(* Logix 5000 project; controller DC01 vendor 1 type 14 code 165 rev 32.12; software revision 32.04; part 7 of 13 *)
(* tags used below, declared in another part *)
   CurrentSchedule : UDT_ShiftString_Breakdown;
   DC1_to_LN02_Messages : DINT[20];
   LN02_Main_Messages : DINT[250];
   LN02_MainLine_MSG_Out : MESSAGE;
   LN02_Schedule : UDT_Current_Status;
   LN02_Theoretical_Units_Counter : COUNTER;
   LN02EHM11 : DINT;
   LN02EJM02 : DINT;
   LN02EJM03 : DINT;
   LN02EKM01 : DINT;
   LN02EKM02 : DINT;
   LN02EKM03 : DINT;
   LN02ELM01 : DINT;
   LN02ELM02 : DINT;
   LN02ELM03 : DINT;
   LN02ELM04 : DINT;
   LN02ELM05 : DINT;
   LN02EMM01 : DINT;
   LN02EMM02 : DINT;
   LN02EMM03 : DINT;
   LN02SKS06 : DINT;
   LN02WHM09 : DINT;
   LN02WHM10 : DINT;
   LN02WJS01 : DINT;
   LN02WJS02 : DINT;
   LN02WJS03 : DINT;
   LN02WKM01 : DINT;
   LN02WKS01 : DINT;
   LN02WKS02 : DINT;
   LN02WKS03 : DINT;
   LN02WKS04 : DINT;
   LN02WKS05 : DINT;
   LN02WLM06 : DINT;
   LN02WLM07 : DINT;
   LN02WMM02 : DINT;
   LN02WMM03 : DINT;
   LN03_DataFromDC1 : DINT[20];
   LN03_Main_Messages : DINT[250];
   LN03_Schedule : UDT_Current_Status;
   LN03_ScheduleUnits_Produced_from_line : DINT;
   LN03_Weekly_Schedule : UDT_Weekly_Schedule;
(* LN02, continued *)

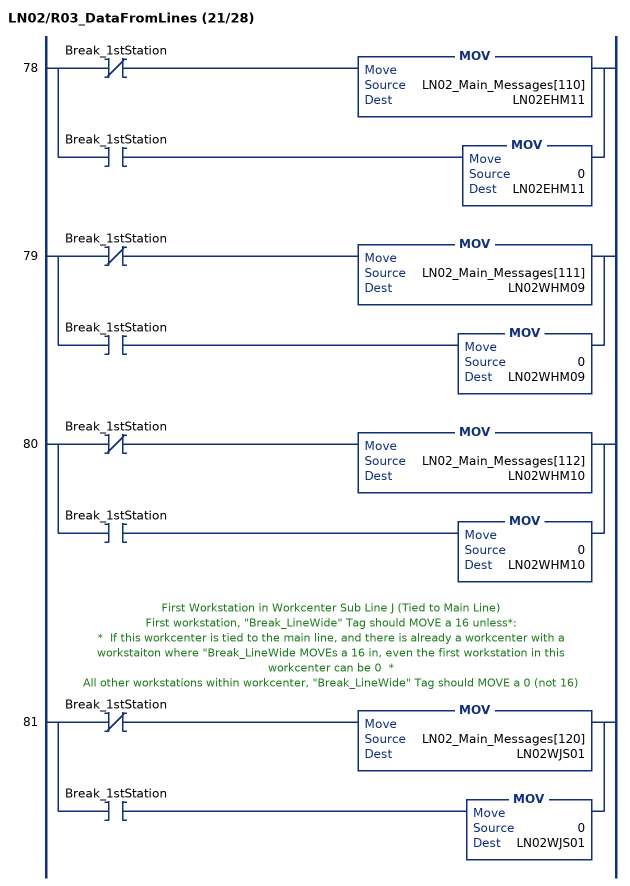
   78: [XIO(Break_1stStation) MOV(LN02_Main_Messages[110],LN02EHM11) ,XIC(Break_1stStation) MOV(0,LN02EHM11) ];
   79: [XIO(Break_1stStation) MOV(LN02_Main_Messages[111],LN02WHM09) ,XIC(Break_1stStation) MOV(0,LN02WHM09) ];
   80: [XIO(Break_1stStation) MOV(LN02_Main_Messages[112],LN02WHM10) ,XIC(Break_1stStation) MOV(0,LN02WHM10) ];
   // First Workstation in Workcenter Sub Line J (Tied to Main Line)
   // First workstation, "Break_LineWide" Tag should MOVE a 16 unless*:
   // *  If this workcenter is tied to the main line, and there is already a workcenter with a workstaiton where "Break_LineWide MOVEs a 16 in, even the first workstation in this workcenter can be 0  *
   // All other workstations within workcenter, "Break_LineWide" Tag should MOVE a 0 (not 16)
   81: [XIO(Break_1stStation) MOV(LN02_Main_Messages[120],LN02WJS01) ,XIC(Break_1stStation) MOV(0,LN02WJS01) ];
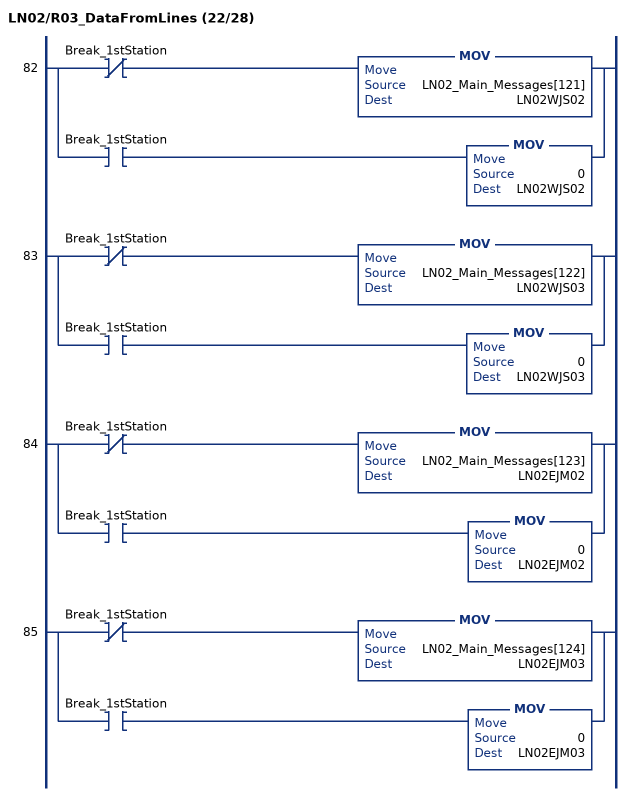
   82: [XIO(Break_1stStation) MOV(LN02_Main_Messages[121],LN02WJS02) ,XIC(Break_1stStation) MOV(0,LN02WJS02) ];
   83: [XIO(Break_1stStation) MOV(LN02_Main_Messages[122],LN02WJS03) ,XIC(Break_1stStation) MOV(0,LN02WJS03) ];
   84: [XIO(Break_1stStation) MOV(LN02_Main_Messages[123],LN02EJM02) ,XIC(Break_1stStation) MOV(0,LN02EJM02) ];
   85: [XIO(Break_1stStation) MOV(LN02_Main_Messages[124],LN02EJM03) ,XIC(Break_1stStation) MOV(0,LN02EJM03) ];
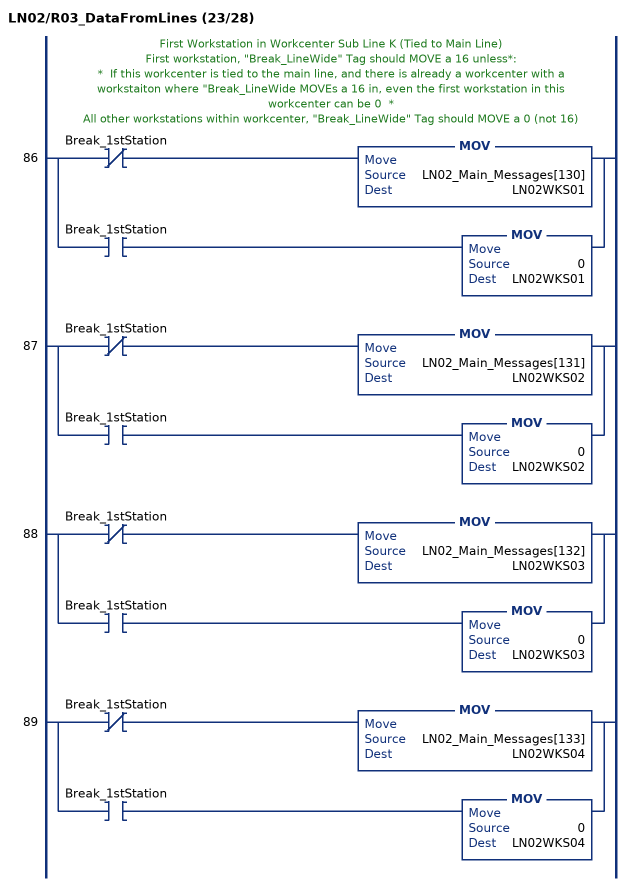
   // First Workstation in Workcenter Sub Line K (Tied to Main Line)
   // First workstation, "Break_LineWide" Tag should MOVE a 16 unless*:
   // *  If this workcenter is tied to the main line, and there is already a workcenter with a workstaiton where "Break_LineWide MOVEs a 16 in, even the first workstation in this workcenter can be 0  *
   // All other workstations within workcenter, "Break_LineWide" Tag should MOVE a 0 (not 16)
   86: [XIO(Break_1stStation) MOV(LN02_Main_Messages[130],LN02WKS01) ,XIC(Break_1stStation) MOV(0,LN02WKS01) ];
   87: [XIO(Break_1stStation) MOV(LN02_Main_Messages[131],LN02WKS02) ,XIC(Break_1stStation) MOV(0,LN02WKS02) ];
   88: [XIO(Break_1stStation) MOV(LN02_Main_Messages[132],LN02WKS03) ,XIC(Break_1stStation) MOV(0,LN02WKS03) ];
   89: [XIO(Break_1stStation) MOV(LN02_Main_Messages[133],LN02WKS04) ,XIC(Break_1stStation) MOV(0,LN02WKS04) ];
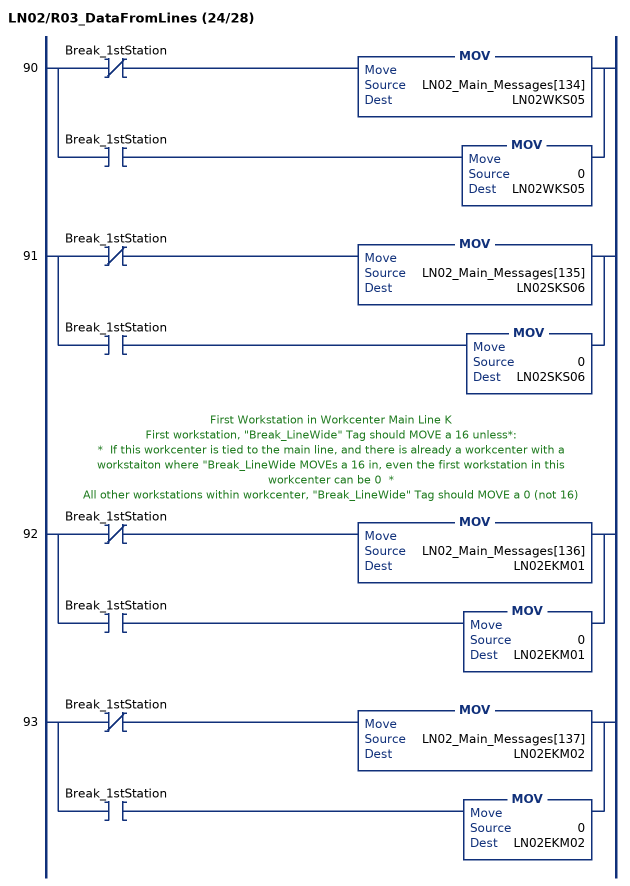
   90: [XIO(Break_1stStation) MOV(LN02_Main_Messages[134],LN02WKS05) ,XIC(Break_1stStation) MOV(0,LN02WKS05) ];
   91: [XIO(Break_1stStation) MOV(LN02_Main_Messages[135],LN02SKS06) ,XIC(Break_1stStation) MOV(0,LN02SKS06) ];
   // First Workstation in Workcenter Main Line K
   // First workstation, "Break_LineWide" Tag should MOVE a 16 unless*:
   // *  If this workcenter is tied to the main line, and there is already a workcenter with a workstaiton where "Break_LineWide MOVEs a 16 in, even the first workstation in this workcenter can be 0  *
   // All other workstations within workcenter, "Break_LineWide" Tag should MOVE a 0 (not 16)
   92: [XIO(Break_1stStation) MOV(LN02_Main_Messages[136],LN02EKM01) ,XIC(Break_1stStation) MOV(0,LN02EKM01) ];
   93: [XIO(Break_1stStation) MOV(LN02_Main_Messages[137],LN02EKM02) ,XIC(Break_1stStation) MOV(0,LN02EKM02) ];
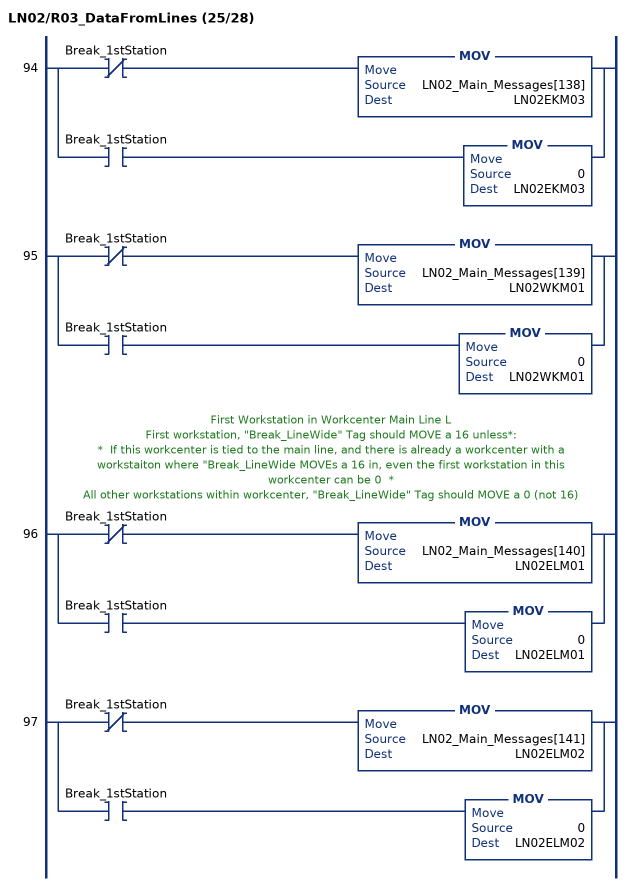
   94: [XIO(Break_1stStation) MOV(LN02_Main_Messages[138],LN02EKM03) ,XIC(Break_1stStation) MOV(0,LN02EKM03) ];
   95: [XIO(Break_1stStation) MOV(LN02_Main_Messages[139],LN02WKM01) ,XIC(Break_1stStation) MOV(0,LN02WKM01) ];
   // First Workstation in Workcenter Main Line L
   // First workstation, "Break_LineWide" Tag should MOVE a 16 unless*:
   // *  If this workcenter is tied to the main line, and there is already a workcenter with a workstaiton where "Break_LineWide MOVEs a 16 in, even the first workstation in this workcenter can be 0  *
   // All other workstations within workcenter, "Break_LineWide" Tag should MOVE a 0 (not 16)
   96: [XIO(Break_1stStation) MOV(LN02_Main_Messages[140],LN02ELM01) ,XIC(Break_1stStation) MOV(0,LN02ELM01) ];
   97: [XIO(Break_1stStation) MOV(LN02_Main_Messages[141],LN02ELM02) ,XIC(Break_1stStation) MOV(0,LN02ELM02) ];
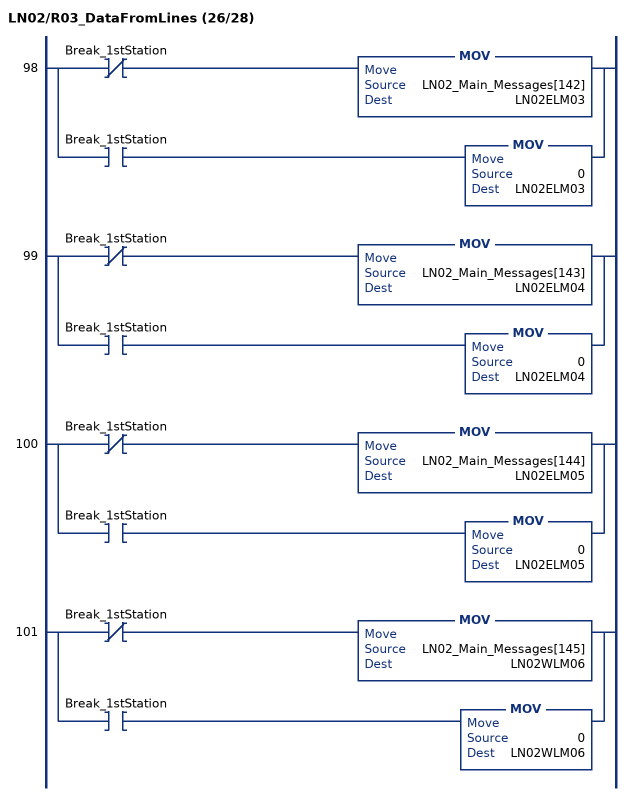
   98: [XIO(Break_1stStation) MOV(LN02_Main_Messages[142],LN02ELM03) ,XIC(Break_1stStation) MOV(0,LN02ELM03) ];
   99: [XIO(Break_1stStation) MOV(LN02_Main_Messages[143],LN02ELM04) ,XIC(Break_1stStation) MOV(0,LN02ELM04) ];
   100: [XIO(Break_1stStation) MOV(LN02_Main_Messages[144],LN02ELM05) ,XIC(Break_1stStation) MOV(0,LN02ELM05) ];
   101: [XIO(Break_1stStation) MOV(LN02_Main_Messages[145],LN02WLM06) ,XIC(Break_1stStation) MOV(0,LN02WLM06) ];
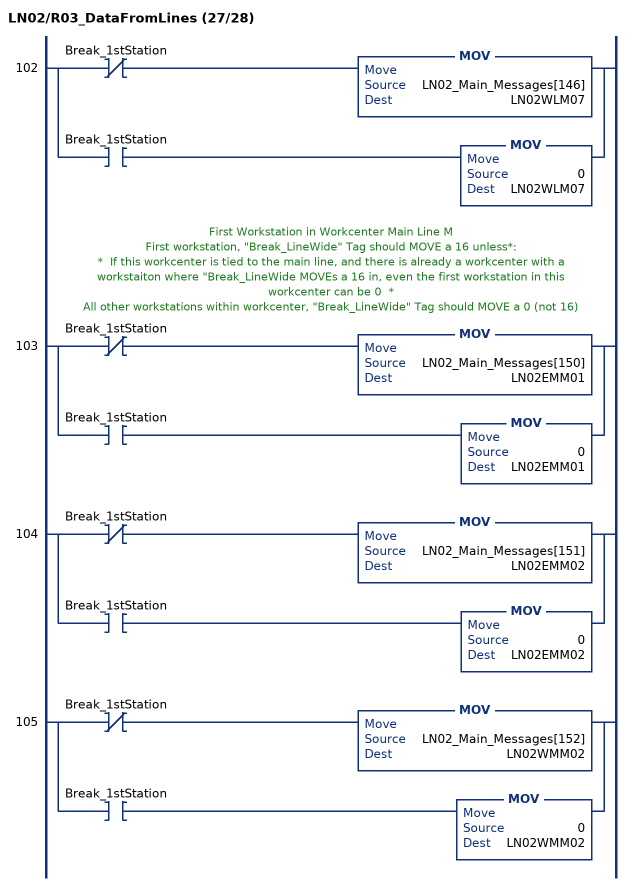
   102: [XIO(Break_1stStation) MOV(LN02_Main_Messages[146],LN02WLM07) ,XIC(Break_1stStation) MOV(0,LN02WLM07) ];
   // First Workstation in Workcenter Main Line M
   // First workstation, "Break_LineWide" Tag should MOVE a 16 unless*:
   // *  If this workcenter is tied to the main line, and there is already a workcenter with a workstaiton where "Break_LineWide MOVEs a 16 in, even the first workstation in this workcenter can be 0  *
   // All other workstations within workcenter, "Break_LineWide" Tag should MOVE a 0 (not 16)
   103: [XIO(Break_1stStation) MOV(LN02_Main_Messages[150],LN02EMM01) ,XIC(Break_1stStation) MOV(0,LN02EMM01) ];
   104: [XIO(Break_1stStation) MOV(LN02_Main_Messages[151],LN02EMM02) ,XIC(Break_1stStation) MOV(0,LN02EMM02) ];
   105: [XIO(Break_1stStation) MOV(LN02_Main_Messages[152],LN02WMM02) ,XIC(Break_1stStation) MOV(0,LN02WMM02) ];
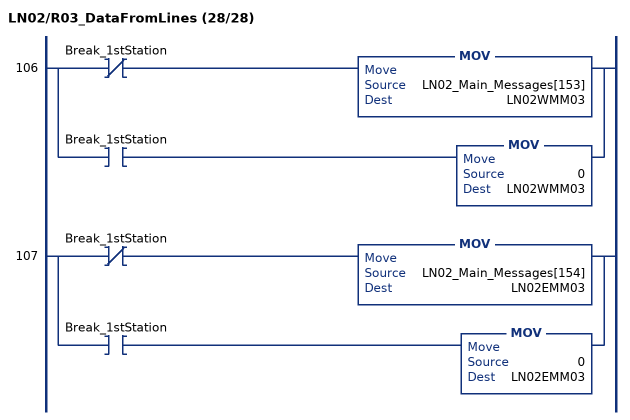
   106: [XIO(Break_1stStation) MOV(LN02_Main_Messages[153],LN02WMM03) ,XIC(Break_1stStation) MOV(0,LN02WMM03) ];
   107: [XIO(Break_1stStation) MOV(LN02_Main_Messages[154],LN02EMM03) ,XIC(Break_1stStation) MOV(0,LN02EMM03) ];
END_ROUTINE

ROUTINE R04_DataToLines   (* ladder *)
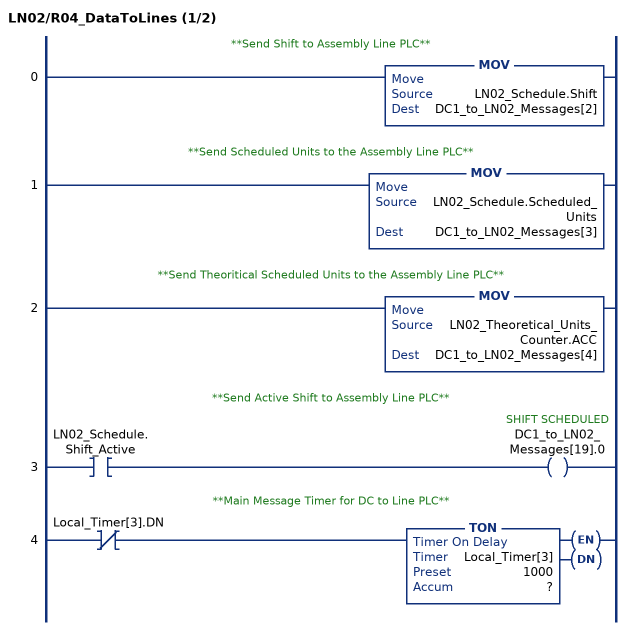
   // **Send Shift to Assembly Line PLC**
   0: MOV(LN02_Schedule.Shift,DC1_to_LN02_Messages[2]);
   // **Send Scheduled Units to the Assembly Line PLC**
   1: MOV(LN02_Schedule.Scheduled_Units,DC1_to_LN02_Messages[3]);
   // **Send Theoritical Scheduled Units to the Assembly Line PLC**
   2: MOV(LN02_Theoretical_Units_Counter.ACC,DC1_to_LN02_Messages[4]);
   // **Send Active Shift to Assembly Line PLC**
   3: XIC(LN02_Schedule.Shift_Active)OTE(DC1_to_LN02_Messages[19].0);
   // **Main Message Timer for DC to Line PLC**
   4: XIO(Local_Timer[3].DN)TON(Local_Timer[3],?,?);
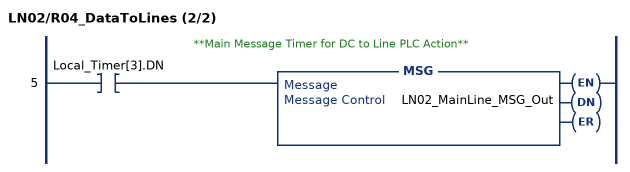
   // **Main Message Timer for DC to Line PLC Action**
   5: XIC(Local_Timer[3].DN)MSG(LN02_MainLine_MSG_Out);
END_ROUTINE
END_PROGRAM

PROGRAM LN03   (* main routine MainRoutine *)
VAR
   Always_Off : BOOL;
   Average_Array : DINT[20];
   Average_Sum : DINT;
   Averaged_LineSpeed : REAL;
   badModel : STRING_40;
   BlockStarveLocal : DINT;
   Break1_Hour : DINT;
   Break1_Hour_String : STRING;
   Break1_Length : DINT;
   Break1_MilliRemain : DINT;
   Break1_Min : DINT;
   Break1_Min_String : STRING;
   Break1_MinDisplay : DINT;
   Break1_SecDisplay : DINT;
   Break1_SecRemain : DINT;
   Break1_SecWholeMin : DINT;
   Break1_Timer : TIMER;
   Break2_Hour : DINT;
   Break2_Hour_String : STRING;
   Break2_Length : DINT;
   Break2_MilliRemain : DINT;
   Break2_Min : DINT;
   Break2_Min_String : STRING;
   Break2_MinDisplay : DINT;
   Break2_SecDisplay : DINT;
   Break2_SecRemain : DINT;
   Break2_SecWholeMin : DINT;
   Break2_Timer : TIMER;
   Break_1stStation : BOOL;
   Break_LineWide : BOOL;
   Break_WorkCenter : BOOL;
   Break_Workstation : BOOL;
   dlw_test : DINT := -805278210;
   End_Hour : DINT := 20;
   End_Hour_String : STRING := '20';
   End_Min : DINT := 3;
   End_Min_String : STRING := '3-';
   faultcount : DINT;
   FaultExists : CONTROL := (LEN := 230, POS := 229, EN := 1, DN := 1);
   firstCharacter : STRING_40 := 'W';
   FlexTimer_HoursDisplay : DINT;
   FlexTimer_MinutesDisplay : DINT;
   FlexTimer_SecondsDisplay : DINT;
   FlexTimertoHours : DINT;
   FlexTimertoMinutes : DINT;
   FlexTimertoSeconds : DINT;
   HoursFromMidnight : DINT;
   HoursFromMidnight_Remain : DINT;
   HoursTilMidnight : DINT;
   HoursTilMidnight_Remain : DINT;
   KnownFaultExist : DINT := 5;
   L02EAS35 : DINT;
   L02EDM16 : DINT;
   LineRate_perSecond_scheduled : DINT;
   LN01_Flex_Timer : TIMER;
   LN01_MainLine_MSG : MESSAGE;
        MessageParameters(ServiceCode := 16#004c, LocalElement := LN03_Main_Messages[0], ...)
   LN01_ML_Message_MSG : MESSAGE;
   LN01_Rotate_Timer : TIMER;
   LN01_SNModel_MSG : MESSAGE;
   LN02EAS35 : DINT;
   LN02EDM16 : DINT;
   LN03_MainLine_MSG : MESSAGE;   // Data Messages From Assembly Line 3 To Data Concentrator 1
        MessageParameters(ServiceCode := 16#004c, LocalElement := LN03_Main_Messages[0], ...)
   Local_Counter : COUNTER[20] := ([0].PRE := 1);
   Local_DATETIME : DINT[20];
   Local_Timer : TIMER[30] := ([0].EN := 1, [0].DN := 1, [3].PRE := 2000, [3].ACC := 1751, [3].EN := 1, [3].TT := 1, [4].PRE := 400, [4].ACC := 391, [4].EN := 1, [4].TT := 1, [6].PRE := 2000, [6].ACC := 150, [6].EN := 1, [6].TT := 1);
   Lunch_Hour : DINT;
   Lunch_Hour_String : STRING;
   Lunch_Length : DINT;
   Lunch_MilliRemain : DINT;
   Lunch_Min : DINT;
   Lunch_Min_String : STRING;
   Lunch_MinDisplay : DINT;
   Lunch_SecDisplay : DINT;
   Lunch_SecRemain : DINT;
   Lunch_SecWholeMin : DINT;
   Lunch_Timer : TIMER;
   Midnight_Hour : DINT;
   mlc_test21 : BOOL;
   null : STRING;
   OneShot : DINT;
   ONS_0 : DINT;
   ONS_20 : DINT;
   prevCalculateLocal : DINT;
   PreviousCount : DINT := 277;
   previousSerialNumber : STRING := 'CA0807422';
   PreviousShift : DINT := 1;
   readIndex : DINT := 41;
   register : DINT := 8;
   Rotate_MilliRemain : DINT;
   Rotate_Seconds_perShift : DINT;
   Rotate_SecRemain : DINT;
   Scheduled_Units_Buffer : DINT := 700;
   Shift_Break_Lengths : DINT;
   Shift_Break_Lengths_Remain : DINT;
   Shift_Delay_Min : DINT := 60;
   Shift_Extra_Min : DINT;
   Shift_Hours : DINT;
   Shift_Hours_Remain : DINT;
   Shift_Minutes : DINT;
   Shift_Minutes_Remain : DINT;
   Shift_Reset : BOOL;
   Shift_Reset_ONS : BOOL := 1;
   Shift_Seconds : DINT;
   Shift_Seconds_Remain : DINT;
   Start_Hour : DINT := 20;
   Start_Hour_String : STRING := '20';
   Start_Min : DINT := 3;
   Start_Min_String : STRING := '3-';
   tempIndex : DINT := 25;
   theoreticalUnitsReal : DINT;
   workstationid : DINT := 250;
   writeIndex : DINT := 42;
END_VAR

ROUTINE MainRoutine   (* ladder *)
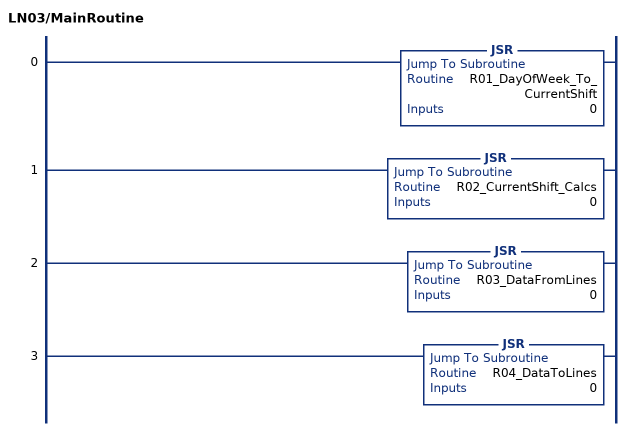
   0: JSR(R01_DayOfWeek_To_CurrentShift,0);
   1: JSR(R02_CurrentShift_Calcs,0);
   2: JSR(R03_DataFromLines,0);
   3: JSR(R04_DataToLines,0);
END_ROUTINE

ROUTINE R01_DayOfWeek_To_CurrentShift   (* ladder *)
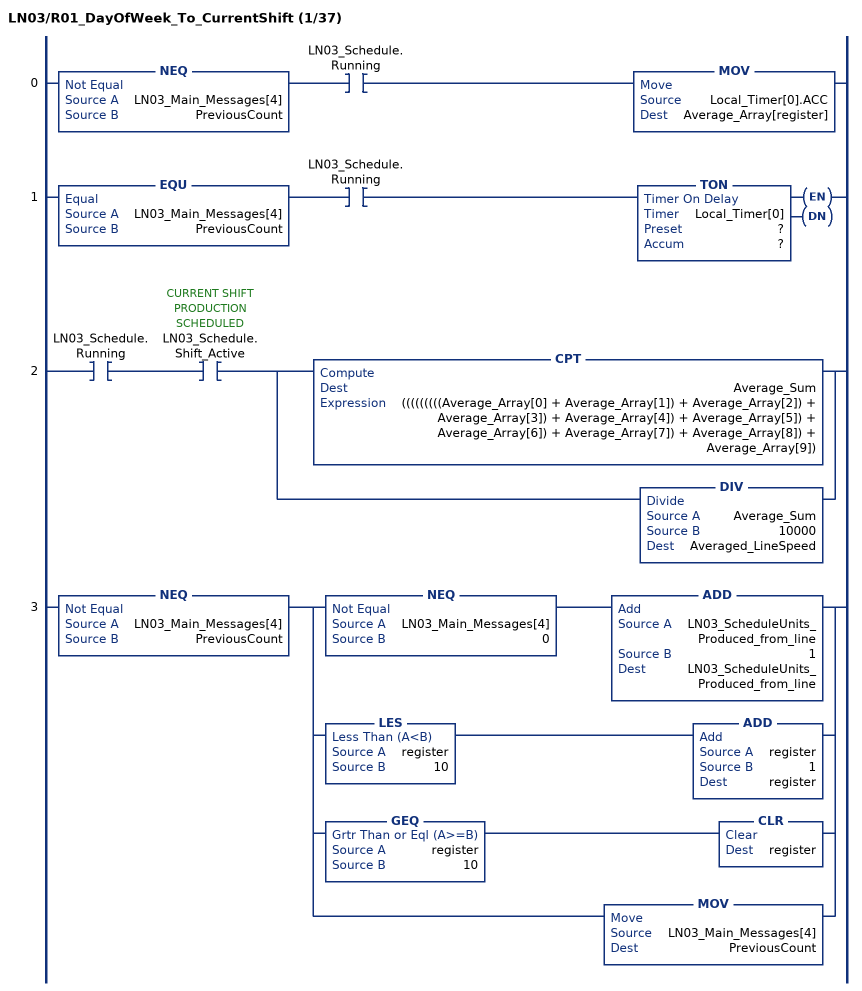
   0: NEQ(LN03_Main_Messages[4],PreviousCount)XIC(LN03_Schedule.Running)MOV(Local_Timer[0].ACC,Average_Array[register]);
   1: EQU(LN03_Main_Messages[4],PreviousCount)XIC(LN03_Schedule.Running)TON(Local_Timer[0],?,?);
   2: XIC(LN03_Schedule.Running)XIC(LN03_Schedule.Shift_Active)[CPT(Average_Sum,(((((((((Average_Array[0] + Average_Array[1]) + Average_Array[2]) + Average_Array[3]) + Average_Array[4]) + Average_Array[5]) + Average_Array[6]) + Average_Array[7]) + Average_Array[8]) + Average_Array[9])) ,DIV(Average_Sum,10000,Averaged_LineSpeed) ];
   3: NEQ(LN03_Main_Messages[4],PreviousCount)[NEQ(LN03_Main_Messages[4],0) ADD(LN03_ScheduleUnits_Produced_from_line,1,LN03_ScheduleUnits_Produced_from_line) ,LES(register,10) ADD(register,1,register) ,GEQ(register,10) CLR(register) ,MOV(LN03_Main_Messages[4],PreviousCount) ];
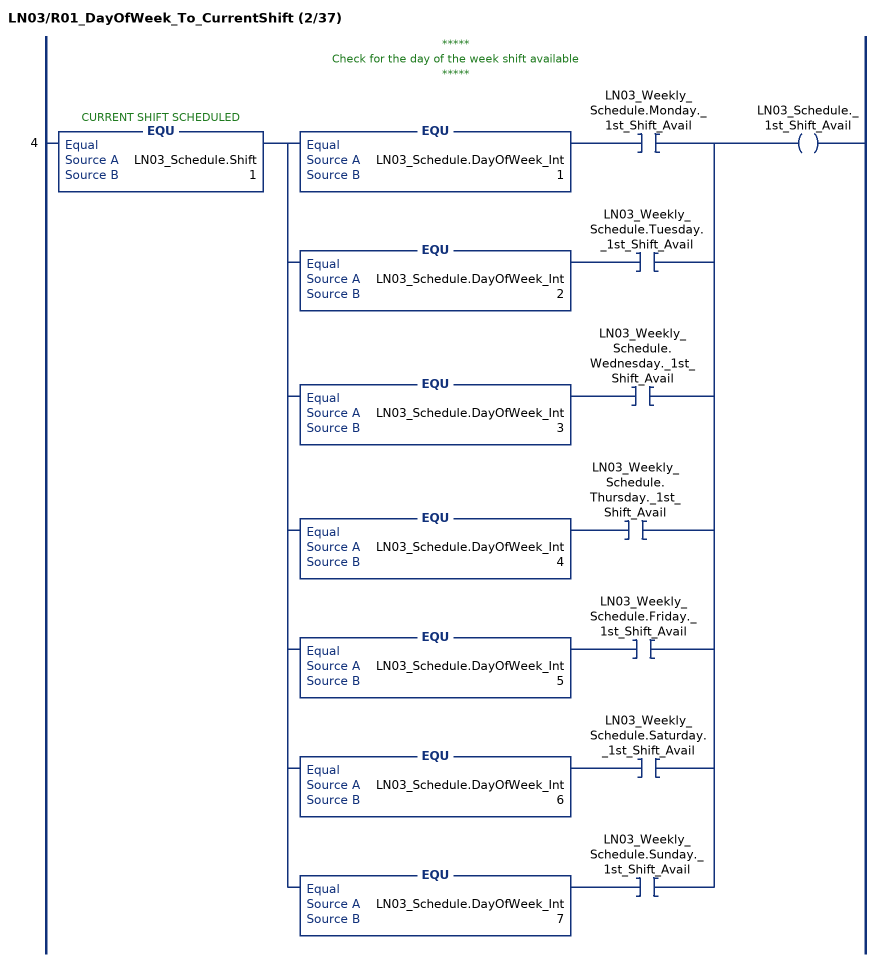
   // *****
   // Check for the day of the week shift available
   // *****
   4: EQU(LN03_Schedule.Shift,1)[EQU(LN03_Schedule.DayOfWeek_Int,1) XIC(LN03_Weekly_Schedule.Monday._1st_Shift_Avail) ,EQU(LN03_Schedule.DayOfWeek_Int,2) XIC(LN03_Weekly_Schedule.Tuesday._1st_Shift_Avail) ,EQU(LN03_Schedule.DayOfWeek_Int,3) XIC(LN03_Weekly_Schedule.Wednesday._1st_Shift_Avail) ,EQU(LN03_Schedule.DayOfWeek_Int,4) XIC(LN03_Weekly_Schedule.Thursday._1st_Shift_Avail) ,EQU(LN03_Schedule.DayOfWeek_Int,5) XIC(LN03_Weekly_Schedule.Friday._1st_Shift_Avail) ,EQU(LN03_Schedule.DayOfWeek_Int,6) XIC(LN03_Weekly_Schedule.Saturday._1st_Shift_Avail) ,EQU(LN03_Schedule.DayOfWeek_Int,7) XIC(LN03_Weekly_Schedule.Sunday._1st_Shift_Avail) ]OTE(LN03_Schedule._1st_Shift_Avail);
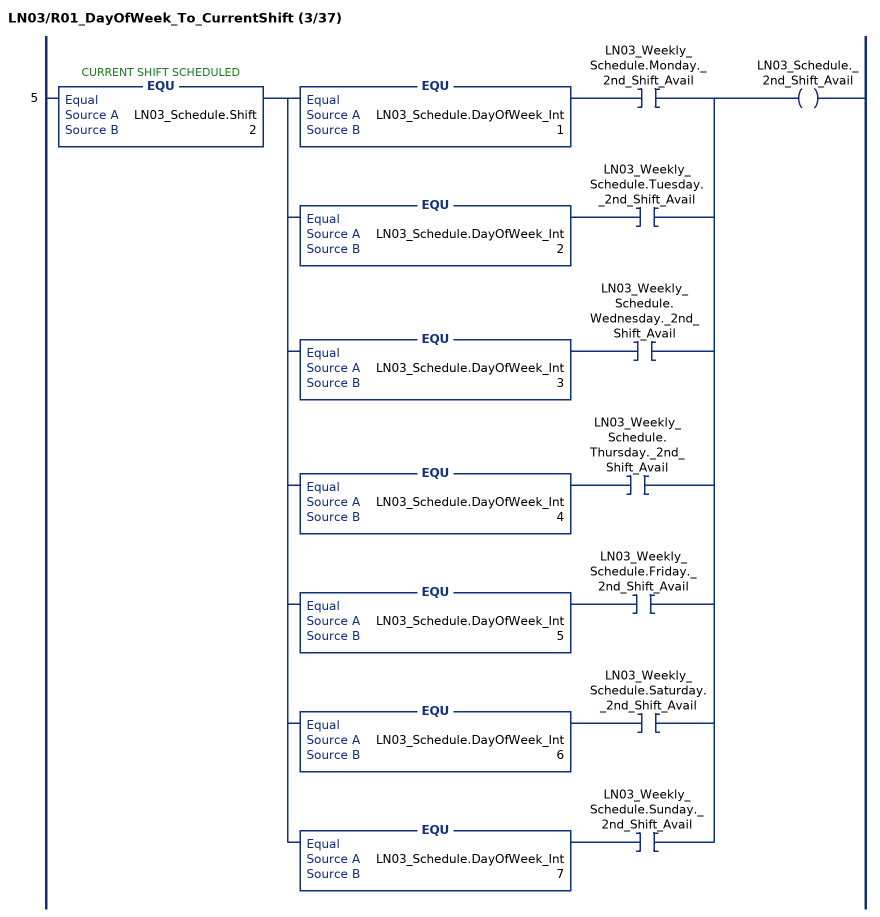
   5: EQU(LN03_Schedule.Shift,2)[EQU(LN03_Schedule.DayOfWeek_Int,1) XIC(LN03_Weekly_Schedule.Monday._2nd_Shift_Avail) ,EQU(LN03_Schedule.DayOfWeek_Int,2) XIC(LN03_Weekly_Schedule.Tuesday._2nd_Shift_Avail) ,EQU(LN03_Schedule.DayOfWeek_Int,3) XIC(LN03_Weekly_Schedule.Wednesday._2nd_Shift_Avail) ,EQU(LN03_Schedule.DayOfWeek_Int,4) XIC(LN03_Weekly_Schedule.Thursday._2nd_Shift_Avail) ,EQU(LN03_Schedule.DayOfWeek_Int,5) XIC(LN03_Weekly_Schedule.Friday._2nd_Shift_Avail) ,EQU(LN03_Schedule.DayOfWeek_Int,6) XIC(LN03_Weekly_Schedule.Saturday._2nd_Shift_Avail) ,EQU(LN03_Schedule.DayOfWeek_Int,7) XIC(LN03_Weekly_Schedule.Sunday._2nd_Shift_Avail) ]OTE(LN03_Schedule._2nd_Shift_Avail);
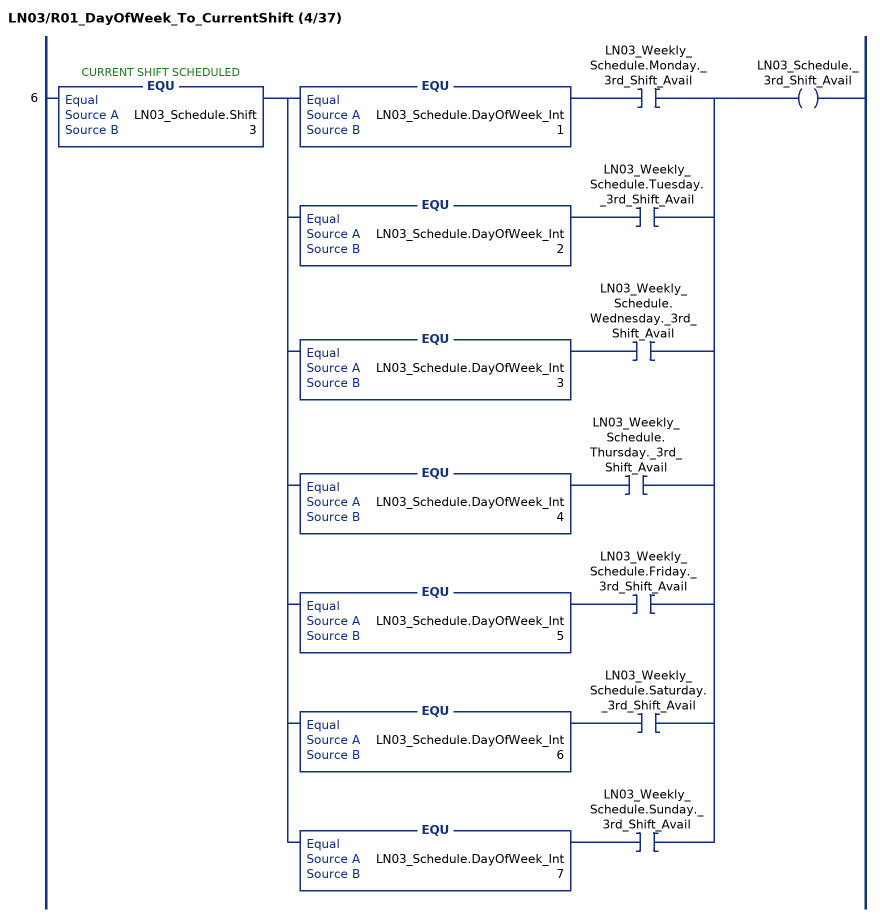
   6: EQU(LN03_Schedule.Shift,3)[EQU(LN03_Schedule.DayOfWeek_Int,1) XIC(LN03_Weekly_Schedule.Monday._3rd_Shift_Avail) ,EQU(LN03_Schedule.DayOfWeek_Int,2) XIC(LN03_Weekly_Schedule.Tuesday._3rd_Shift_Avail) ,EQU(LN03_Schedule.DayOfWeek_Int,3) XIC(LN03_Weekly_Schedule.Wednesday._3rd_Shift_Avail) ,EQU(LN03_Schedule.DayOfWeek_Int,4) XIC(LN03_Weekly_Schedule.Thursday._3rd_Shift_Avail) ,EQU(LN03_Schedule.DayOfWeek_Int,5) XIC(LN03_Weekly_Schedule.Friday._3rd_Shift_Avail) ,EQU(LN03_Schedule.DayOfWeek_Int,6) XIC(LN03_Weekly_Schedule.Saturday._3rd_Shift_Avail) ,EQU(LN03_Schedule.DayOfWeek_Int,7) XIC(LN03_Weekly_Schedule.Sunday._3rd_Shift_Avail) ]OTE(LN03_Schedule._3rd_Shift_Avail);
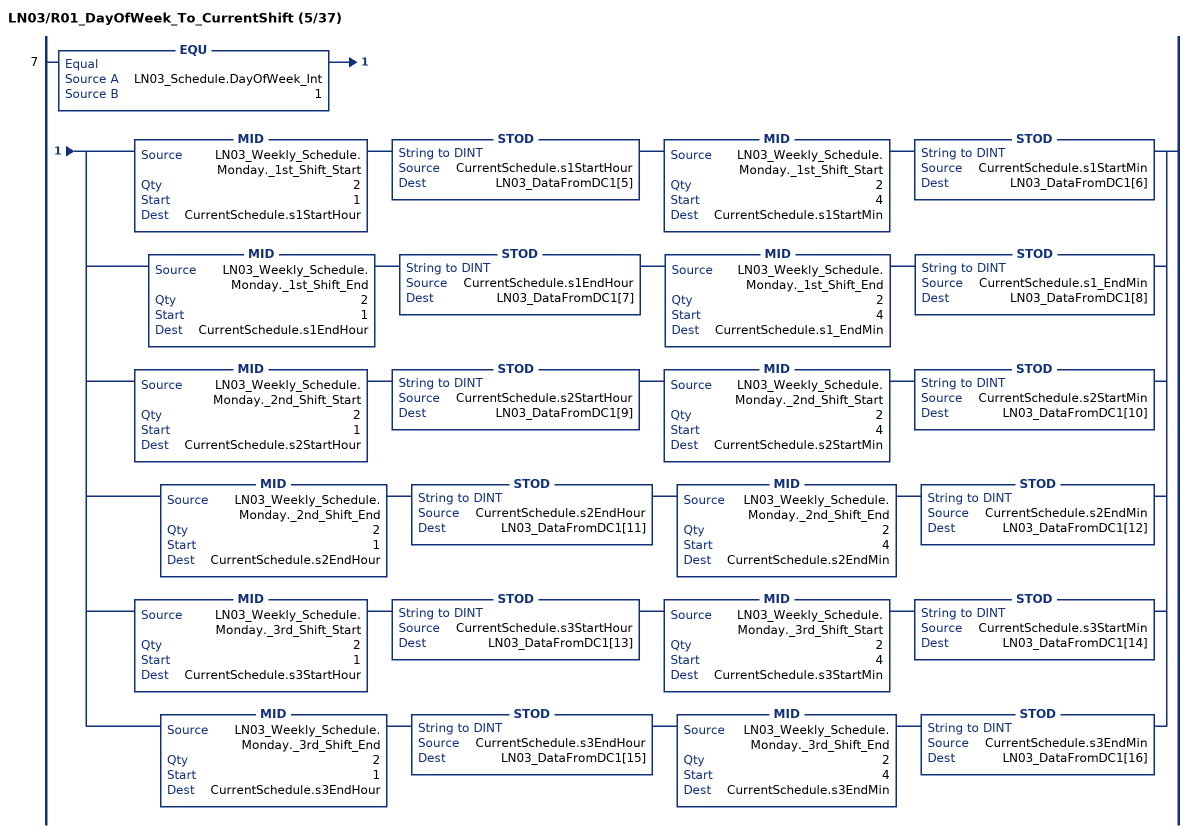
   7: EQU(LN03_Schedule.DayOfWeek_Int,1)[MID(LN03_Weekly_Schedule.Monday._1st_Shift_Start,2,1,CurrentSchedule.s1StartHour) STOD(CurrentSchedule.s1StartHour,LN03_DataFromDC1[5]) MID(LN03_Weekly_Schedule.Monday._1st_Shift_Start,2,4,CurrentSchedule.s1StartMin) STOD(CurrentSchedule.s1StartMin,LN03_DataFromDC1[6]) ,MID(LN03_Weekly_Schedule.Monday._1st_Shift_End,2,1,CurrentSchedule.s1EndHour) STOD(CurrentSchedule.s1EndHour,LN03_DataFromDC1[7]) MID(LN03_Weekly_Schedule.Monday._1st_Shift_End,2,4,CurrentSchedule.s1_EndMin) STOD(CurrentSchedule.s1_EndMin,LN03_DataFromDC1[8]) ,MID(LN03_Weekly_Schedule.Monday._2nd_Shift_Start,2,1,CurrentSchedule.s2StartHour) STOD(CurrentSchedule.s2StartHour,LN03_DataFromDC1[9]) MID(LN03_Weekly_Schedule.Monday._2nd_Shift_Start,2,4,CurrentSchedule.s2StartMin) STOD(CurrentSchedule.s2StartMin,LN03_DataFromDC1[10]) ,MID(LN03_Weekly_Schedule.Monday._2nd_Shift_End,2,1,CurrentSchedule.s2EndHour) STOD(CurrentSchedule.s2EndHour,LN03_DataFromDC1[11]) MID(LN03_Weekly_Schedule.Monday._2nd_Shift_End,2,4,CurrentSchedule.s2EndMin) STOD(CurrentSchedule.s2EndMin,LN03_DataFromDC1[12]) ,MID(LN03_Weekly_Schedule.Monday._3rd_Shift_Start,2,1,CurrentSchedule.s3StartHour) STOD(CurrentSchedule.s3StartHour,LN03_DataFromDC1[13]) MID(LN03_Weekly_Schedule.Monday._3rd_Shift_Start,2,4,CurrentSchedule.s3StartMin) STOD(CurrentSchedule.s3StartMin,LN03_DataFromDC1[14]) ,MID(LN03_Weekly_Schedule.Monday._3rd_Shift_End,2,1,CurrentSchedule.s3EndHour) STOD(CurrentSchedule.s3EndHour,LN03_DataFromDC1[15]) MID(LN03_Weekly_Schedule.Monday._3rd_Shift_End,2,4,CurrentSchedule.s3EndMin) STOD(CurrentSchedule.s3EndMin,LN03_DataFromDC1[16]) ];
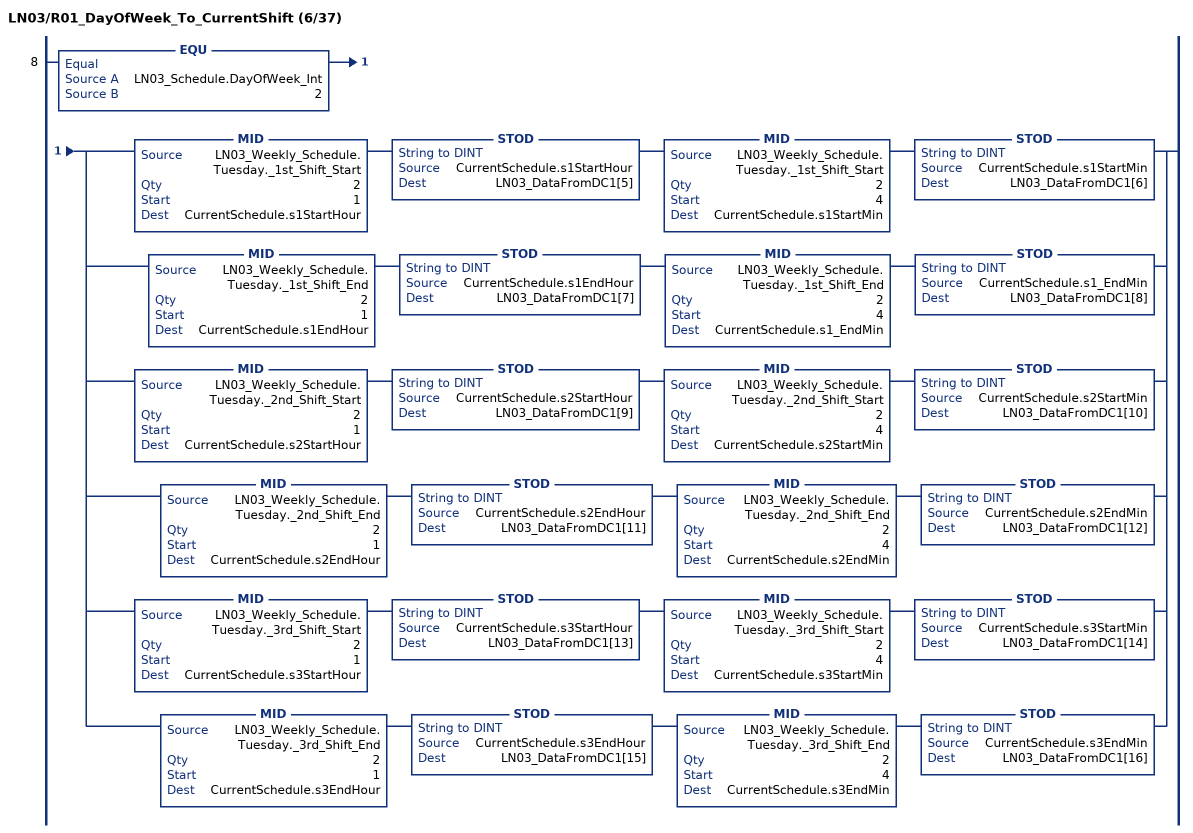
   8: EQU(LN03_Schedule.DayOfWeek_Int,2)[MID(LN03_Weekly_Schedule.Tuesday._1st_Shift_Start,2,1,CurrentSchedule.s1StartHour) STOD(CurrentSchedule.s1StartHour,LN03_DataFromDC1[5]) MID(LN03_Weekly_Schedule.Tuesday._1st_Shift_Start,2,4,CurrentSchedule.s1StartMin) STOD(CurrentSchedule.s1StartMin,LN03_DataFromDC1[6]) ,MID(LN03_Weekly_Schedule.Tuesday._1st_Shift_End,2,1,CurrentSchedule.s1EndHour) STOD(CurrentSchedule.s1EndHour,LN03_DataFromDC1[7]) MID(LN03_Weekly_Schedule.Tuesday._1st_Shift_End,2,4,CurrentSchedule.s1_EndMin) STOD(CurrentSchedule.s1_EndMin,LN03_DataFromDC1[8]) ,MID(LN03_Weekly_Schedule.Tuesday._2nd_Shift_Start,2,1,CurrentSchedule.s2StartHour) STOD(CurrentSchedule.s2StartHour,LN03_DataFromDC1[9]) MID(LN03_Weekly_Schedule.Tuesday._2nd_Shift_Start,2,4,CurrentSchedule.s2StartMin) STOD(CurrentSchedule.s2StartMin,LN03_DataFromDC1[10]) ,MID(LN03_Weekly_Schedule.Tuesday._2nd_Shift_End,2,1,CurrentSchedule.s2EndHour) STOD(CurrentSchedule.s2EndHour,LN03_DataFromDC1[11]) MID(LN03_Weekly_Schedule.Tuesday._2nd_Shift_End,2,4,CurrentSchedule.s2EndMin) STOD(CurrentSchedule.s2EndMin,LN03_DataFromDC1[12]) ,MID(LN03_Weekly_Schedule.Tuesday._3rd_Shift_Start,2,1,CurrentSchedule.s3StartHour) STOD(CurrentSchedule.s3StartHour,LN03_DataFromDC1[13]) MID(LN03_Weekly_Schedule.Tuesday._3rd_Shift_Start,2,4,CurrentSchedule.s3StartMin) STOD(CurrentSchedule.s3StartMin,LN03_DataFromDC1[14]) ,MID(LN03_Weekly_Schedule.Tuesday._3rd_Shift_End,2,1,CurrentSchedule.s3EndHour) STOD(CurrentSchedule.s3EndHour,LN03_DataFromDC1[15]) MID(LN03_Weekly_Schedule.Tuesday._3rd_Shift_End,2,4,CurrentSchedule.s3EndMin) STOD(CurrentSchedule.s3EndMin,LN03_DataFromDC1[16]) ];
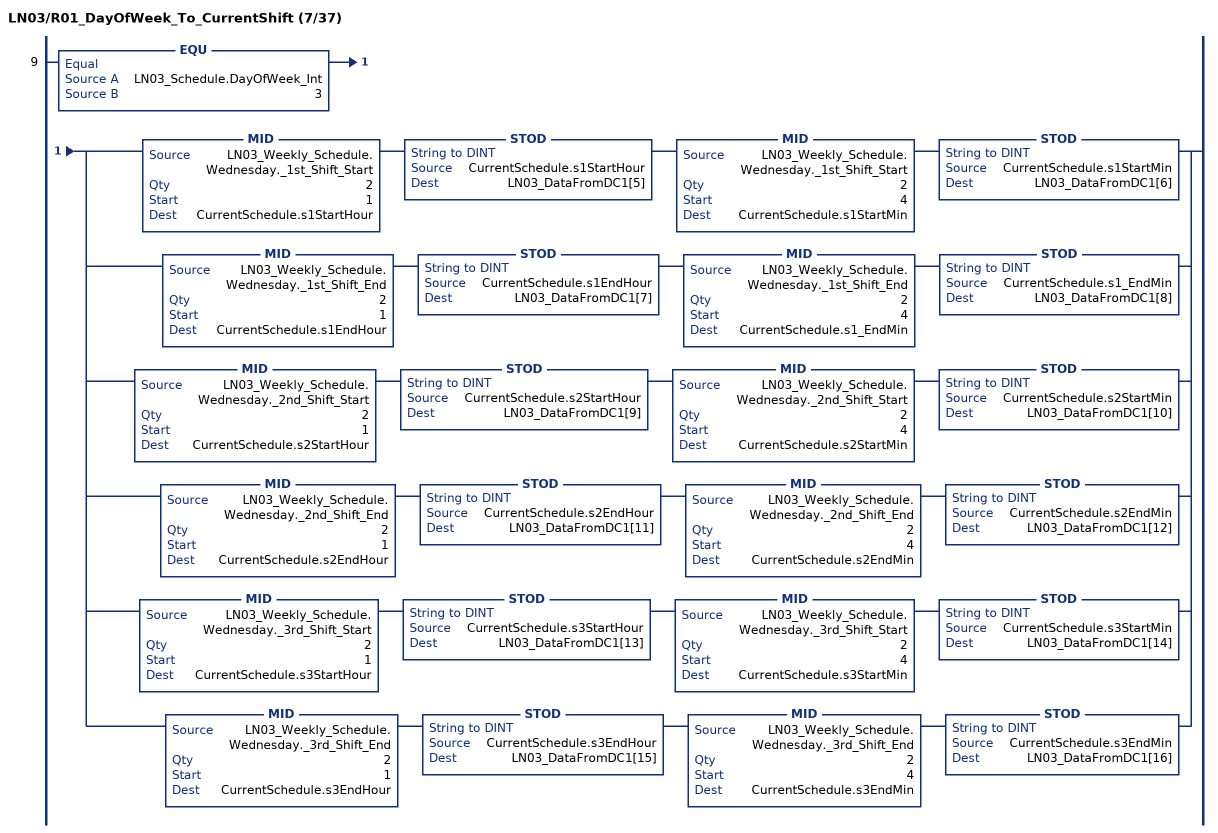
   9: EQU(LN03_Schedule.DayOfWeek_Int,3)[MID(LN03_Weekly_Schedule.Wednesday._1st_Shift_Start,2,1,CurrentSchedule.s1StartHour) STOD(CurrentSchedule.s1StartHour,LN03_DataFromDC1[5]) MID(LN03_Weekly_Schedule.Wednesday._1st_Shift_Start,2,4,CurrentSchedule.s1StartMin) STOD(CurrentSchedule.s1StartMin,LN03_DataFromDC1[6]) ,MID(LN03_Weekly_Schedule.Wednesday._1st_Shift_End,2,1,CurrentSchedule.s1EndHour) STOD(CurrentSchedule.s1EndHour,LN03_DataFromDC1[7]) MID(LN03_Weekly_Schedule.Wednesday._1st_Shift_End,2,4,CurrentSchedule.s1_EndMin) STOD(CurrentSchedule.s1_EndMin,LN03_DataFromDC1[8]) ,MID(LN03_Weekly_Schedule.Wednesday._2nd_Shift_Start,2,1,CurrentSchedule.s2StartHour) STOD(CurrentSchedule.s2StartHour,LN03_DataFromDC1[9]) MID(LN03_Weekly_Schedule.Wednesday._2nd_Shift_Start,2,4,CurrentSchedule.s2StartMin) STOD(CurrentSchedule.s2StartMin,LN03_DataFromDC1[10]) ,MID(LN03_Weekly_Schedule.Wednesday._2nd_Shift_End,2,1,CurrentSchedule.s2EndHour) STOD(CurrentSchedule.s2EndHour,LN03_DataFromDC1[11]) MID(LN03_Weekly_Schedule.Wednesday._2nd_Shift_End,2,4,CurrentSchedule.s2EndMin) STOD(CurrentSchedule.s2EndMin,LN03_DataFromDC1[12]) ,MID(LN03_Weekly_Schedule.Wednesday._3rd_Shift_Start,2,1,CurrentSchedule.s3StartHour) STOD(CurrentSchedule.s3StartHour,LN03_DataFromDC1[13]) MID(LN03_Weekly_Schedule.Wednesday._3rd_Shift_Start,2,4,CurrentSchedule.s3StartMin) STOD(CurrentSchedule.s3StartMin,LN03_DataFromDC1[14]) ,MID(LN03_Weekly_Schedule.Wednesday._3rd_Shift_End,2,1,CurrentSchedule.s3EndHour) STOD(CurrentSchedule.s3EndHour,LN03_DataFromDC1[15]) MID(LN03_Weekly_Schedule.Wednesday._3rd_Shift_End,2,4,CurrentSchedule.s3EndMin) STOD(CurrentSchedule.s3EndMin,LN03_DataFromDC1[16]) ];
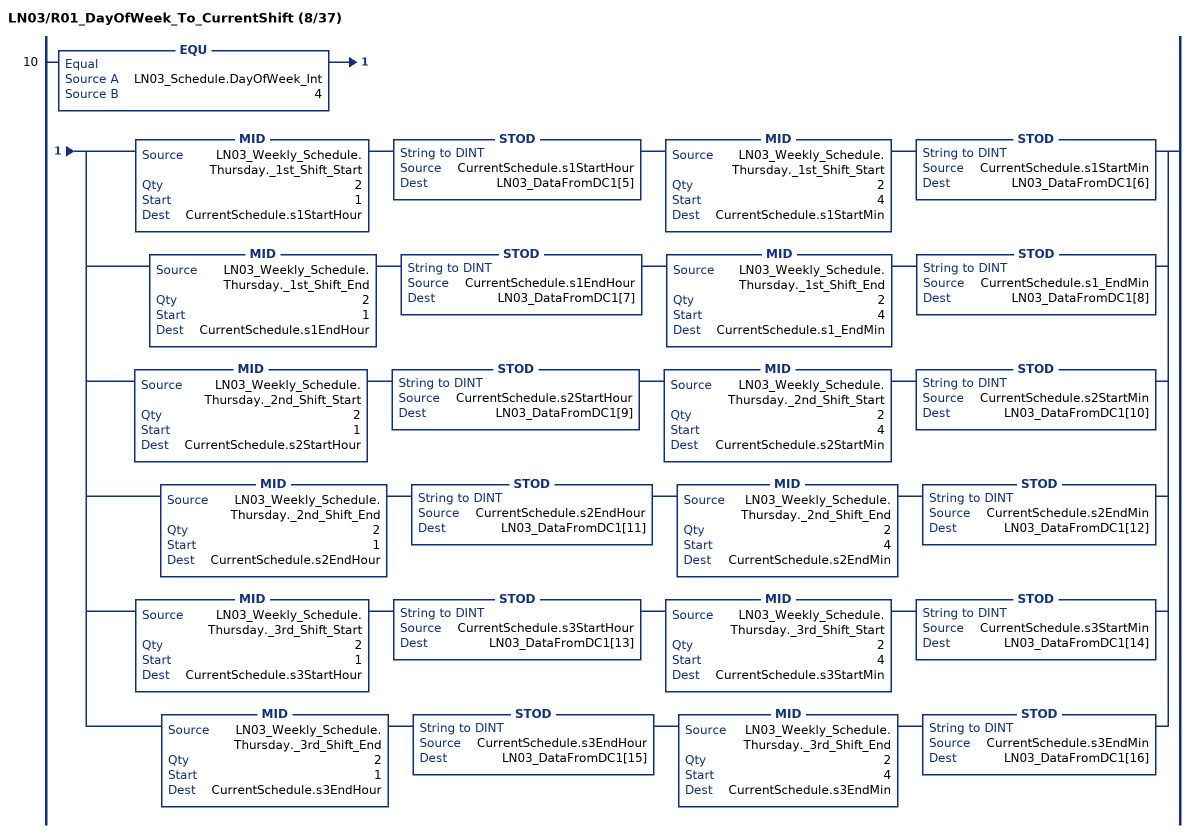
   10: EQU(LN03_Schedule.DayOfWeek_Int,4)[MID(LN03_Weekly_Schedule.Thursday._1st_Shift_Start,2,1,CurrentSchedule.s1StartHour) STOD(CurrentSchedule.s1StartHour,LN03_DataFromDC1[5]) MID(LN03_Weekly_Schedule.Thursday._1st_Shift_Start,2,4,CurrentSchedule.s1StartMin) STOD(CurrentSchedule.s1StartMin,LN03_DataFromDC1[6]) ,MID(LN03_Weekly_Schedule.Thursday._1st_Shift_End,2,1,CurrentSchedule.s1EndHour) STOD(CurrentSchedule.s1EndHour,LN03_DataFromDC1[7]) MID(LN03_Weekly_Schedule.Thursday._1st_Shift_End,2,4,CurrentSchedule.s1_EndMin) STOD(CurrentSchedule.s1_EndMin,LN03_DataFromDC1[8]) ,MID(LN03_Weekly_Schedule.Thursday._2nd_Shift_Start,2,1,CurrentSchedule.s2StartHour) STOD(CurrentSchedule.s2StartHour,LN03_DataFromDC1[9]) MID(LN03_Weekly_Schedule.Thursday._2nd_Shift_Start,2,4,CurrentSchedule.s2StartMin) STOD(CurrentSchedule.s2StartMin,LN03_DataFromDC1[10]) ,MID(LN03_Weekly_Schedule.Thursday._2nd_Shift_End,2,1,CurrentSchedule.s2EndHour) STOD(CurrentSchedule.s2EndHour,LN03_DataFromDC1[11]) MID(LN03_Weekly_Schedule.Thursday._2nd_Shift_End,2,4,CurrentSchedule.s2EndMin) STOD(CurrentSchedule.s2EndMin,LN03_DataFromDC1[12]) ,MID(LN03_Weekly_Schedule.Thursday._3rd_Shift_Start,2,1,CurrentSchedule.s3StartHour) STOD(CurrentSchedule.s3StartHour,LN03_DataFromDC1[13]) MID(LN03_Weekly_Schedule.Thursday._3rd_Shift_Start,2,4,CurrentSchedule.s3StartMin) STOD(CurrentSchedule.s3StartMin,LN03_DataFromDC1[14]) ,MID(LN03_Weekly_Schedule.Thursday._3rd_Shift_End,2,1,CurrentSchedule.s3EndHour) STOD(CurrentSchedule.s3EndHour,LN03_DataFromDC1[15]) MID(LN03_Weekly_Schedule.Thursday._3rd_Shift_End,2,4,CurrentSchedule.s3EndMin) STOD(CurrentSchedule.s3EndMin,LN03_DataFromDC1[16]) ];
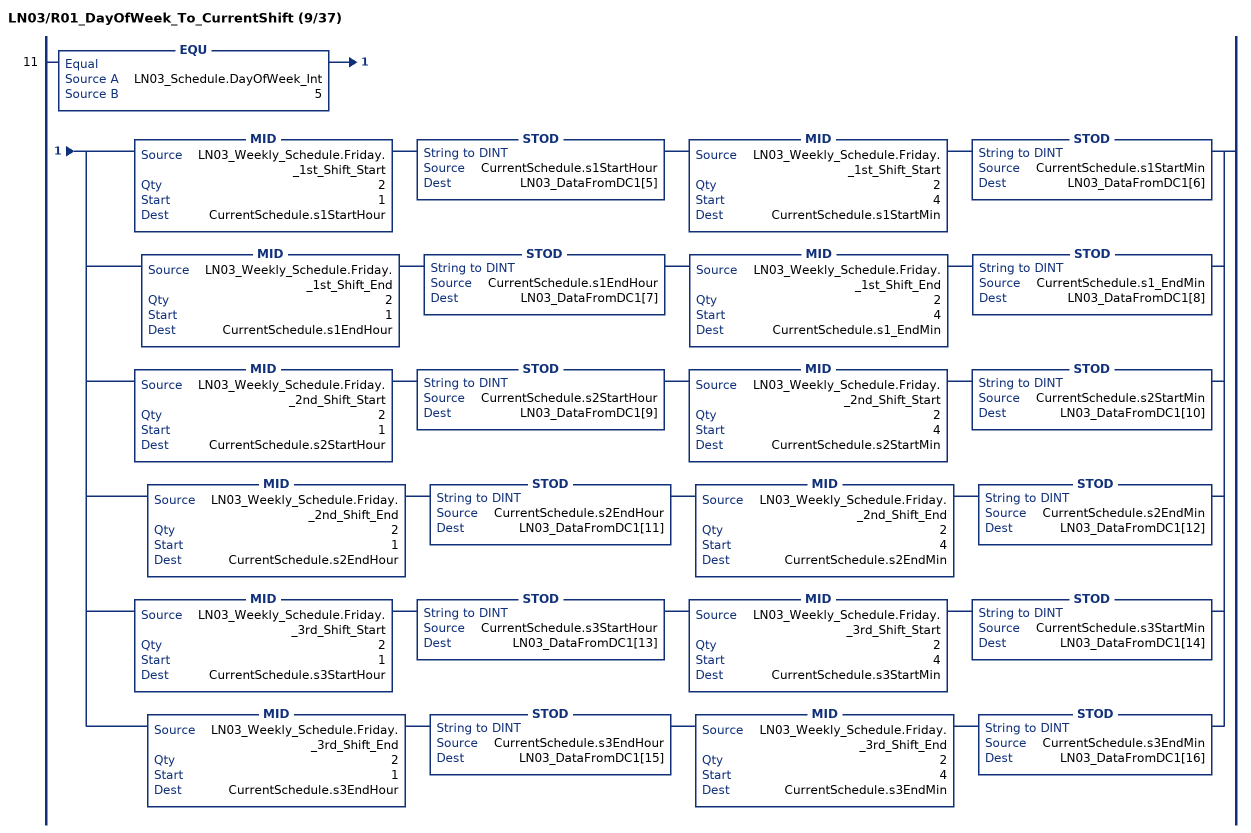
   11: EQU(LN03_Schedule.DayOfWeek_Int,5)[MID(LN03_Weekly_Schedule.Friday._1st_Shift_Start,2,1,CurrentSchedule.s1StartHour) STOD(CurrentSchedule.s1StartHour,LN03_DataFromDC1[5]) MID(LN03_Weekly_Schedule.Friday._1st_Shift_Start,2,4,CurrentSchedule.s1StartMin) STOD(CurrentSchedule.s1StartMin,LN03_DataFromDC1[6]) ,MID(LN03_Weekly_Schedule.Friday._1st_Shift_End,2,1,CurrentSchedule.s1EndHour) STOD(CurrentSchedule.s1EndHour,LN03_DataFromDC1[7]) MID(LN03_Weekly_Schedule.Friday._1st_Shift_End,2,4,CurrentSchedule.s1_EndMin) STOD(CurrentSchedule.s1_EndMin,LN03_DataFromDC1[8]) ,MID(LN03_Weekly_Schedule.Friday._2nd_Shift_Start,2,1,CurrentSchedule.s2StartHour) STOD(CurrentSchedule.s2StartHour,LN03_DataFromDC1[9]) MID(LN03_Weekly_Schedule.Friday._2nd_Shift_Start,2,4,CurrentSchedule.s2StartMin) STOD(CurrentSchedule.s2StartMin,LN03_DataFromDC1[10]) ,MID(LN03_Weekly_Schedule.Friday._2nd_Shift_End,2,1,CurrentSchedule.s2EndHour) STOD(CurrentSchedule.s2EndHour,LN03_DataFromDC1[11]) MID(LN03_Weekly_Schedule.Friday._2nd_Shift_End,2,4,CurrentSchedule.s2EndMin) STOD(CurrentSchedule.s2EndMin,LN03_DataFromDC1[12]) ,MID(LN03_Weekly_Schedule.Friday._3rd_Shift_Start,2,1,CurrentSchedule.s3StartHour) STOD(CurrentSchedule.s3StartHour,LN03_DataFromDC1[13]) MID(LN03_Weekly_Schedule.Friday._3rd_Shift_Start,2,4,CurrentSchedule.s3StartMin) STOD(CurrentSchedule.s3StartMin,LN03_DataFromDC1[14]) ,MID(LN03_Weekly_Schedule.Friday._3rd_Shift_End,2,1,CurrentSchedule.s3EndHour) STOD(CurrentSchedule.s3EndHour,LN03_DataFromDC1[15]) MID(LN03_Weekly_Schedule.Friday._3rd_Shift_End,2,4,CurrentSchedule.s3EndMin) STOD(CurrentSchedule.s3EndMin,LN03_DataFromDC1[16]) ];
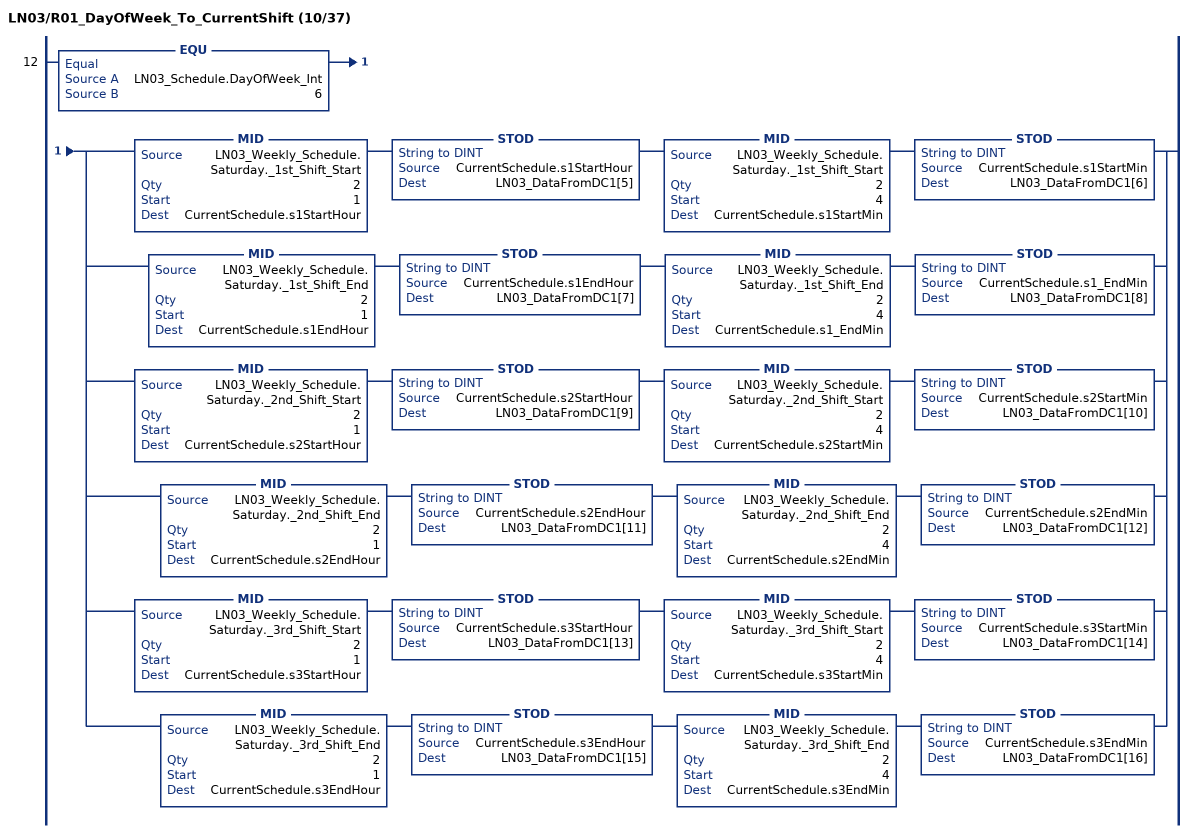
   12: EQU(LN03_Schedule.DayOfWeek_Int,6)[MID(LN03_Weekly_Schedule.Saturday._1st_Shift_Start,2,1,CurrentSchedule.s1StartHour) STOD(CurrentSchedule.s1StartHour,LN03_DataFromDC1[5]) MID(LN03_Weekly_Schedule.Saturday._1st_Shift_Start,2,4,CurrentSchedule.s1StartMin) STOD(CurrentSchedule.s1StartMin,LN03_DataFromDC1[6]) ,MID(LN03_Weekly_Schedule.Saturday._1st_Shift_End,2,1,CurrentSchedule.s1EndHour) STOD(CurrentSchedule.s1EndHour,LN03_DataFromDC1[7]) MID(LN03_Weekly_Schedule.Saturday._1st_Shift_End,2,4,CurrentSchedule.s1_EndMin) STOD(CurrentSchedule.s1_EndMin,LN03_DataFromDC1[8]) ,MID(LN03_Weekly_Schedule.Saturday._2nd_Shift_Start,2,1,CurrentSchedule.s2StartHour) STOD(CurrentSchedule.s2StartHour,LN03_DataFromDC1[9]) MID(LN03_Weekly_Schedule.Saturday._2nd_Shift_Start,2,4,CurrentSchedule.s2StartMin) STOD(CurrentSchedule.s2StartMin,LN03_DataFromDC1[10]) ,MID(LN03_Weekly_Schedule.Saturday._2nd_Shift_End,2,1,CurrentSchedule.s2EndHour) STOD(CurrentSchedule.s2EndHour,LN03_DataFromDC1[11]) MID(LN03_Weekly_Schedule.Saturday._2nd_Shift_End,2,4,CurrentSchedule.s2EndMin) STOD(CurrentSchedule.s2EndMin,LN03_DataFromDC1[12]) ,MID(LN03_Weekly_Schedule.Saturday._3rd_Shift_Start,2,1,CurrentSchedule.s3StartHour) STOD(CurrentSchedule.s3StartHour,LN03_DataFromDC1[13]) MID(LN03_Weekly_Schedule.Saturday._3rd_Shift_Start,2,4,CurrentSchedule.s3StartMin) STOD(CurrentSchedule.s3StartMin,LN03_DataFromDC1[14]) ,MID(LN03_Weekly_Schedule.Saturday._3rd_Shift_End,2,1,CurrentSchedule.s3EndHour) STOD(CurrentSchedule.s3EndHour,LN03_DataFromDC1[15]) MID(LN03_Weekly_Schedule.Saturday._3rd_Shift_End,2,4,CurrentSchedule.s3EndMin) STOD(CurrentSchedule.s3EndMin,LN03_DataFromDC1[16]) ];
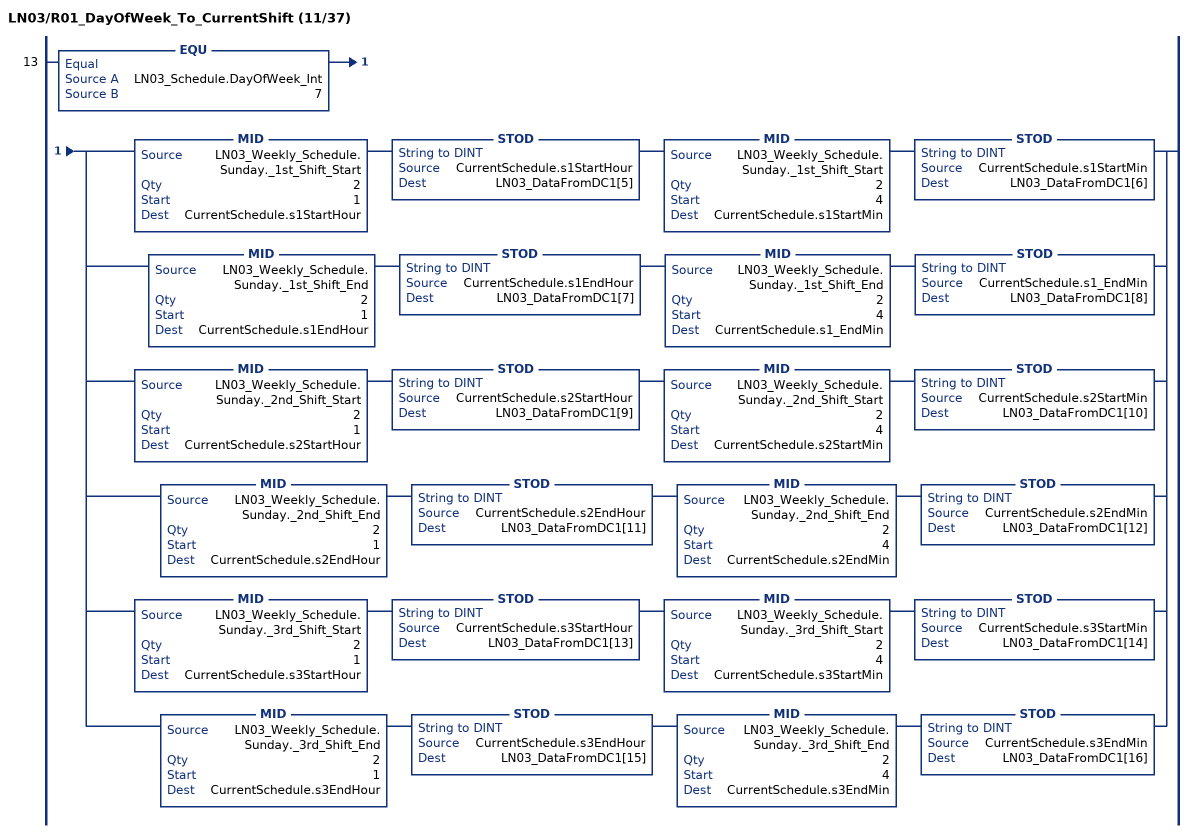
   13: EQU(LN03_Schedule.DayOfWeek_Int,7)[MID(LN03_Weekly_Schedule.Sunday._1st_Shift_Start,2,1,CurrentSchedule.s1StartHour) STOD(CurrentSchedule.s1StartHour,LN03_DataFromDC1[5]) MID(LN03_Weekly_Schedule.Sunday._1st_Shift_Start,2,4,CurrentSchedule.s1StartMin) STOD(CurrentSchedule.s1StartMin,LN03_DataFromDC1[6]) ,MID(LN03_Weekly_Schedule.Sunday._1st_Shift_End,2,1,CurrentSchedule.s1EndHour) STOD(CurrentSchedule.s1EndHour,LN03_DataFromDC1[7]) MID(LN03_Weekly_Schedule.Sunday._1st_Shift_End,2,4,CurrentSchedule.s1_EndMin) STOD(CurrentSchedule.s1_EndMin,LN03_DataFromDC1[8]) ,MID(LN03_Weekly_Schedule.Sunday._2nd_Shift_Start,2,1,CurrentSchedule.s2StartHour) STOD(CurrentSchedule.s2StartHour,LN03_DataFromDC1[9]) MID(LN03_Weekly_Schedule.Sunday._2nd_Shift_Start,2,4,CurrentSchedule.s2StartMin) STOD(CurrentSchedule.s2StartMin,LN03_DataFromDC1[10]) ,MID(LN03_Weekly_Schedule.Sunday._2nd_Shift_End,2,1,CurrentSchedule.s2EndHour) STOD(CurrentSchedule.s2EndHour,LN03_DataFromDC1[11]) MID(LN03_Weekly_Schedule.Sunday._2nd_Shift_End,2,4,CurrentSchedule.s2EndMin) STOD(CurrentSchedule.s2EndMin,LN03_DataFromDC1[12]) ,MID(LN03_Weekly_Schedule.Sunday._3rd_Shift_Start,2,1,CurrentSchedule.s3StartHour) STOD(CurrentSchedule.s3StartHour,LN03_DataFromDC1[13]) MID(LN03_Weekly_Schedule.Sunday._3rd_Shift_Start,2,4,CurrentSchedule.s3StartMin) STOD(CurrentSchedule.s3StartMin,LN03_DataFromDC1[14]) ,MID(LN03_Weekly_Schedule.Sunday._3rd_Shift_End,2,1,CurrentSchedule.s3EndHour) STOD(CurrentSchedule.s3EndHour,LN03_DataFromDC1[15]) MID(LN03_Weekly_Schedule.Sunday._3rd_Shift_End,2,4,CurrentSchedule.s3EndMin) STOD(CurrentSchedule.s3EndMin,LN03_DataFromDC1[16]) ];
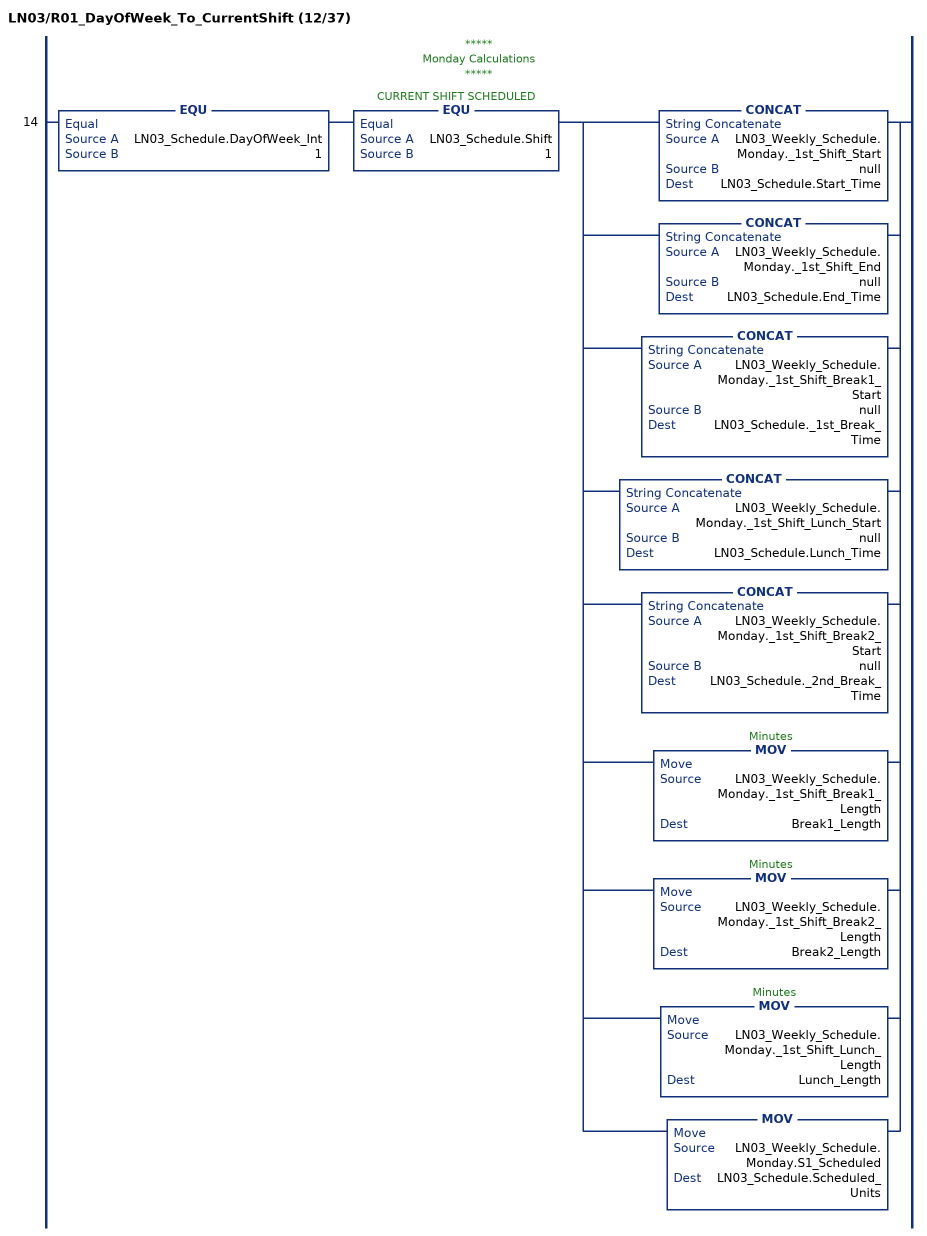
   // *****
   // Monday Calculations
   // *****
   14: EQU(LN03_Schedule.DayOfWeek_Int,1)EQU(LN03_Schedule.Shift,1)[CONCAT(LN03_Weekly_Schedule.Monday._1st_Shift_Start,null,LN03_Schedule.Start_Time) ,CONCAT(LN03_Weekly_Schedule.Monday._1st_Shift_End,null,LN03_Schedule.End_Time) ,CONCAT(LN03_Weekly_Schedule.Monday._1st_Shift_Break1_Start,null,LN03_Schedule._1st_Break_Time) ,CONCAT(LN03_Weekly_Schedule.Monday._1st_Shift_Lunch_Start,null,LN03_Schedule.Lunch_Time) ,CONCAT(LN03_Weekly_Schedule.Monday._1st_Shift_Break2_Start,null,LN03_Schedule._2nd_Break_Time) ,MOV(LN03_Weekly_Schedule.Monday._1st_Shift_Break1_Length,Break1_Length) ,MOV(LN03_Weekly_Schedule.Monday._1st_Shift_Break2_Length,Break2_Length) ,MOV(LN03_Weekly_Schedule.Monday._1st_Shift_Lunch_Length,Lunch_Length) ,MOV(LN03_Weekly_Schedule.Monday.S1_Scheduled,LN03_Schedule.Scheduled_Units) ];
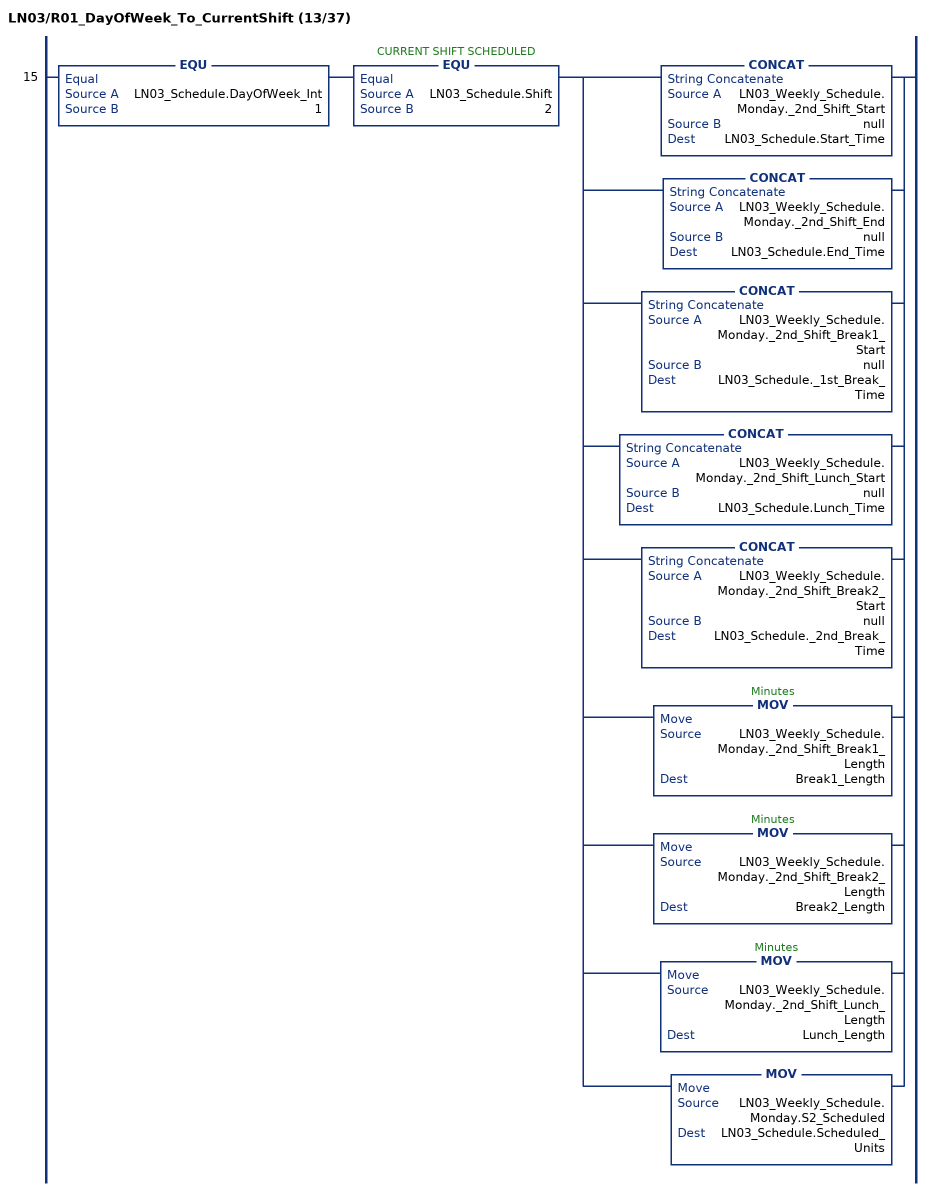
   15: EQU(LN03_Schedule.DayOfWeek_Int,1)EQU(LN03_Schedule.Shift,2)[CONCAT(LN03_Weekly_Schedule.Monday._2nd_Shift_Start,null,LN03_Schedule.Start_Time) ,CONCAT(LN03_Weekly_Schedule.Monday._2nd_Shift_End,null,LN03_Schedule.End_Time) ,CONCAT(LN03_Weekly_Schedule.Monday._2nd_Shift_Break1_Start,null,LN03_Schedule._1st_Break_Time) ,CONCAT(LN03_Weekly_Schedule.Monday._2nd_Shift_Lunch_Start,null,LN03_Schedule.Lunch_Time) ,CONCAT(LN03_Weekly_Schedule.Monday._2nd_Shift_Break2_Start,null,LN03_Schedule._2nd_Break_Time) ,MOV(LN03_Weekly_Schedule.Monday._2nd_Shift_Break1_Length,Break1_Length) ,MOV(LN03_Weekly_Schedule.Monday._2nd_Shift_Break2_Length,Break2_Length) ,MOV(LN03_Weekly_Schedule.Monday._2nd_Shift_Lunch_Length,Lunch_Length) ,MOV(LN03_Weekly_Schedule.Monday.S2_Scheduled,LN03_Schedule.Scheduled_Units) ];
